// SIMATIC S7-200 SMART project (STEP 7-Micro/WIN SMART), CPU ST40

SYMBOL_TABLE 表格 1
MODBUS_INC       VW100
END_SYMBOL_TABLE

SYMBOL_TABLE 系统符号
Always_On        SM0.0    // 始终接通
END_SYMBOL_TABLE

ORGANIZATION_BLOCK MAIN:OB1
TITLE=程序注释
BEGIN
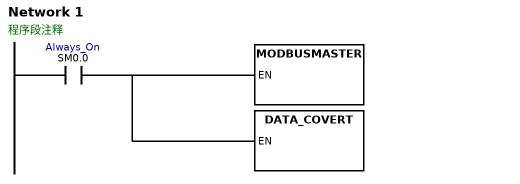
Network 1
// 程序段注释
LD     Always_On:SM0.0
CALL   MODBUSMASTER:SBR41
CALL   DATA_COVERT:SBR4
END_ORGANIZATION_BLOCK

// SBR1: protected block, not included

// SBR2: protected block, not included

// SBR3: protected block, not included

SUBROUTINE_BLOCK DATA_COVERT:SBR4
TITLE=子程序注释
BEGIN
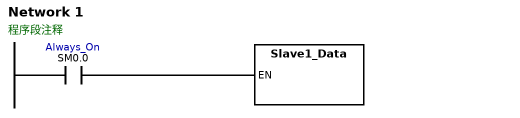
Network 1
// 程序段注释
LD     Always_On:SM0.0
CALL   Slave1_Data:SBR5
END_SUBROUTINE_BLOCK

SUBROUTINE_BLOCK Int_Float:SBR6
TITLE=子程序注释
VAR_INPUT
INPUT:INT;	// LW0 
Coefficient:REAL;	// LD2 
END_VAR
VAR_OUTPUT
OUTPUT:REAL;	// LD6 
END_VAR
VAR
DINT_TEMP:DINT;	// LD10 
REAL_TEMP:REAL;	// LD14 
END_VAR
BEGIN
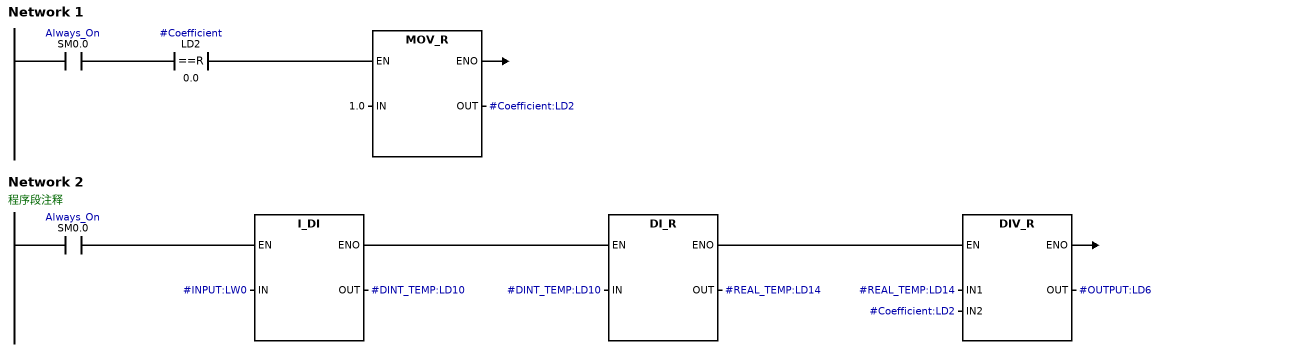
Network 1
LD     Always_On:SM0.0
AR=    #Coefficient:LD2, 0.0
MOVR   1.0, #Coefficient:LD2
Network 2
// 程序段注释
LD     Always_On:SM0.0
ITD    #INPUT:LW0, #DINT_TEMP:LD10
AENO
DTR    #DINT_TEMP:LD10, #REAL_TEMP:LD14
AENO
MOVR   #REAL_TEMP:LD14, #OUTPUT:LD6
/R     #Coefficient:LD2, #OUTPUT:LD6
END_SUBROUTINE_BLOCK

SUBROUTINE_BLOCK Dint_Float:SBR7
TITLE=
VAR_INPUT
INPUT:INT;	// LW0 
Coefficient:REAL;	// LD2 
END_VAR
VAR_OUTPUT
OUT_PUT:REAL;	// LD6 
END_VAR
VAR
DINT_TEMP:DINT;	// LD10 
REAL_TEMP:REAL;	// LD14 
END_VAR
BEGIN
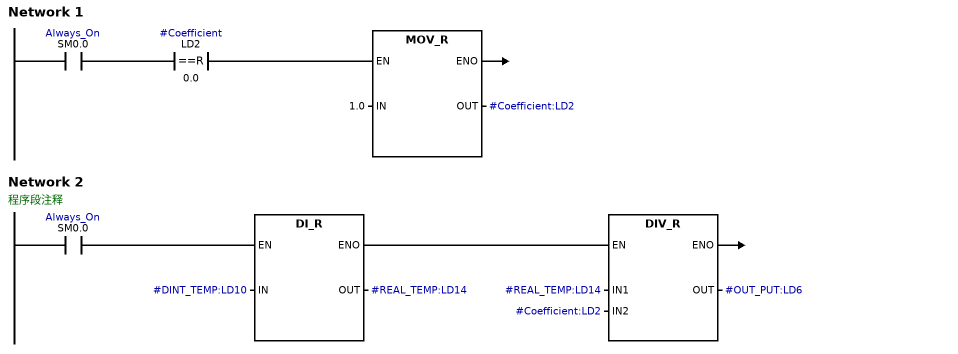
Network 1
LD     Always_On:SM0.0
AR=    #Coefficient:LD2, 0.0
MOVR   1.0, #Coefficient:LD2
Network 2
// 程序段注释
LD     Always_On:SM0.0
DTR    #DINT_TEMP:LD10, #REAL_TEMP:LD14
AENO
MOVR   #REAL_TEMP:LD14, #OUT_PUT:LD6
/R     #Coefficient:LD2, #OUT_PUT:LD6
END_SUBROUTINE_BLOCK

SUBROUTINE_BLOCK MODBUSMASTER:SBR41
TITLE=
VAR
TEMP:BYTE;	// LB0 
TEMP1:BYTE;	// LB1 
TEMP2:BYTE;	// LB2 
TEMP3:BYTE;	// LB3 
TEMP4:BYTE;	// LB4 
TEMP5:BYTE;	// LB5 
TEMP6:BYTE;	// LB6 
TEMPBIT:BOOL;	// L7.0 
TEMPBIT1:BOOL;	// L7.1 
TEMPBIT2:BOOL;	// L7.2 
TEMPBIT3:BOOL;	// L7.3 
TEMPBIT4:BOOL;	// L7.4 
TEMPBIT5:BOOL;	// L7.5 
TEMPBIT6:BOOL;	// L7.6 
END_VAR
BEGIN
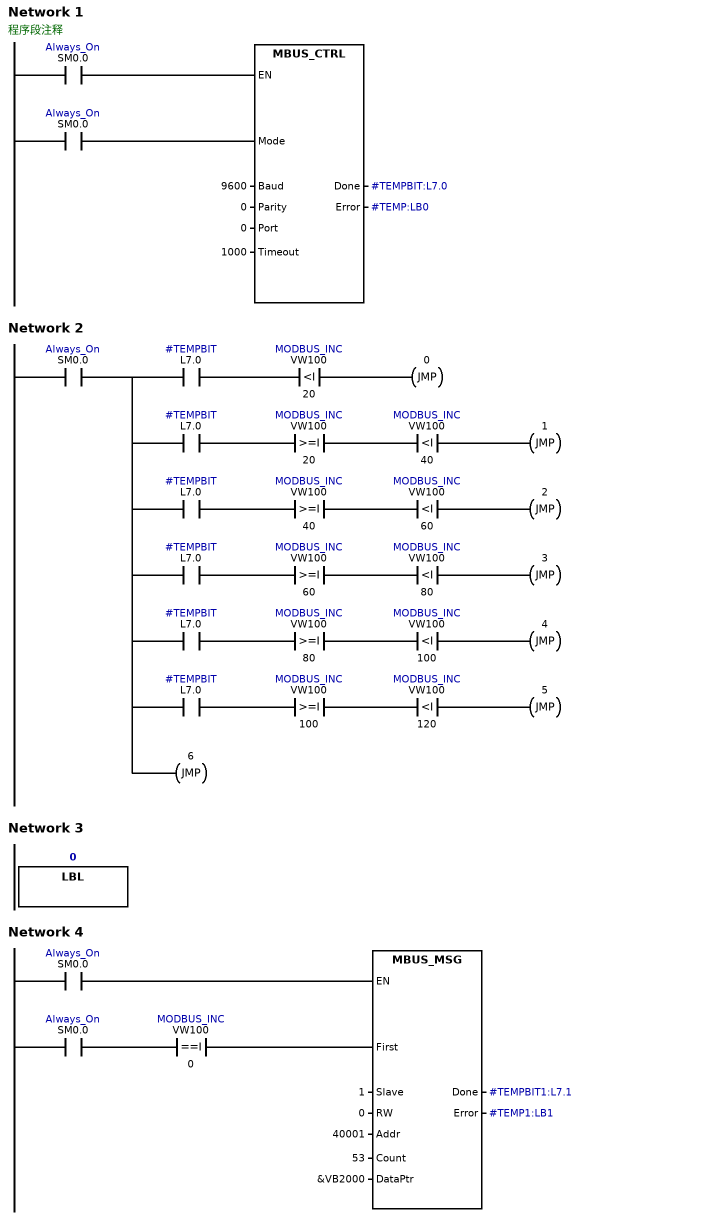
Network 1
// 程序段注释
LD     Always_On:SM0.0
=      L60.0
LD     Always_On:SM0.0
=      L63.7
LD     L60.0
CALL   MBUS_CTRL:SBR1, L63.7, 9600, 0, 0, 1000, #TEMPBIT:L7.0, #TEMP:LB0
Network 2
LD     Always_On:SM0.0
LPS
A      #TEMPBIT:L7.0
AW<    MODBUS_INC:VW100, 20
JMP    0
LRD
A      #TEMPBIT:L7.0
AW>=   MODBUS_INC:VW100, 20
AW<    MODBUS_INC:VW100, 40
JMP    1
LRD
A      #TEMPBIT:L7.0
AW>=   MODBUS_INC:VW100, 40
AW<    MODBUS_INC:VW100, 60
JMP    2
LRD
A      #TEMPBIT:L7.0
AW>=   MODBUS_INC:VW100, 60
AW<    MODBUS_INC:VW100, 80
JMP    3
LRD
A      #TEMPBIT:L7.0
AW>=   MODBUS_INC:VW100, 80
AW<    MODBUS_INC:VW100, 100
JMP    4
LRD
A      #TEMPBIT:L7.0
AW>=   MODBUS_INC:VW100, 100
AW<    MODBUS_INC:VW100, 120
JMP    5
LPP
JMP    6
Network 3
LBL    0
Network 4
LD     Always_On:SM0.0
=      L60.0
LD     Always_On:SM0.0
AW=    MODBUS_INC:VW100, 0
=      L63.7
LD     L60.0
CALL   MBUS_MSG:SBR2, L63.7, 1, 0, 40001, 53, &VB2000, #TEMPBIT1:L7.1, #TEMP1:LB1
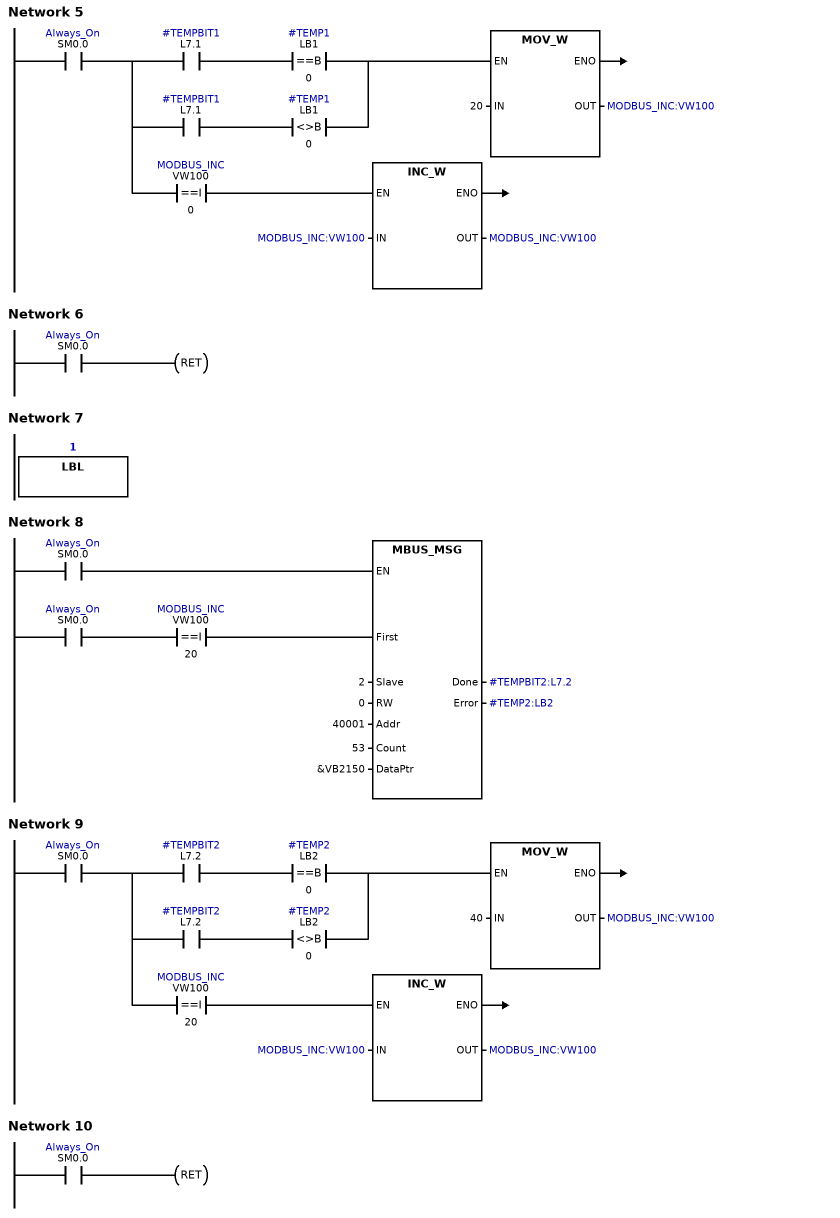
Network 5
LD     Always_On:SM0.0
LPS
LD     #TEMPBIT1:L7.1
AB=    #TEMP1:LB1, 0
LD     #TEMPBIT1:L7.1
AB<>   #TEMP1:LB1, 0
OLD
ALD
MOVW   20, MODBUS_INC:VW100
LPP
AW=    MODBUS_INC:VW100, 0
INCW   MODBUS_INC:VW100
Network 6
LD     Always_On:SM0.0
CRET
Network 7
LBL    1
Network 8
LD     Always_On:SM0.0
=      L60.0
LD     Always_On:SM0.0
AW=    MODBUS_INC:VW100, 20
=      L63.7
LD     L60.0
CALL   MBUS_MSG:SBR2, L63.7, 2, 0, 40001, 53, &VB2150, #TEMPBIT2:L7.2, #TEMP2:LB2
Network 9
LD     Always_On:SM0.0
LPS
LD     #TEMPBIT2:L7.2
AB=    #TEMP2:LB2, 0
LD     #TEMPBIT2:L7.2
AB<>   #TEMP2:LB2, 0
OLD
ALD
MOVW   40, MODBUS_INC:VW100
LPP
AW=    MODBUS_INC:VW100, 20
INCW   MODBUS_INC:VW100
Network 10
LD     Always_On:SM0.0
CRET
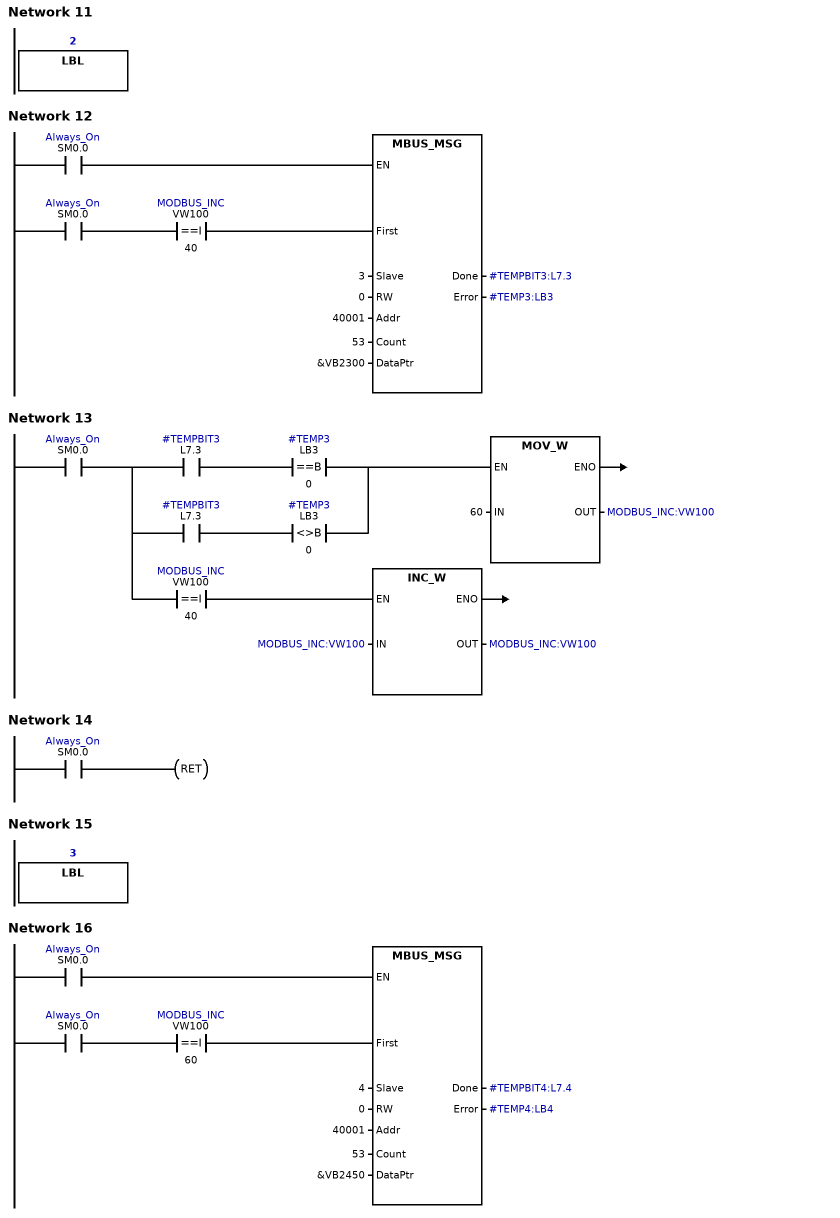
Network 11
LBL    2
Network 12
LD     Always_On:SM0.0
=      L60.0
LD     Always_On:SM0.0
AW=    MODBUS_INC:VW100, 40
=      L63.7
LD     L60.0
CALL   MBUS_MSG:SBR2, L63.7, 3, 0, 40001, 53, &VB2300, #TEMPBIT3:L7.3, #TEMP3:LB3
Network 13
LD     Always_On:SM0.0
LPS
LD     #TEMPBIT3:L7.3
AB=    #TEMP3:LB3, 0
LD     #TEMPBIT3:L7.3
AB<>   #TEMP3:LB3, 0
OLD
ALD
MOVW   60, MODBUS_INC:VW100
LPP
AW=    MODBUS_INC:VW100, 40
INCW   MODBUS_INC:VW100
Network 14
LD     Always_On:SM0.0
CRET
Network 15
LBL    3
Network 16
LD     Always_On:SM0.0
=      L60.0
LD     Always_On:SM0.0
AW=    MODBUS_INC:VW100, 60
=      L63.7
LD     L60.0
CALL   MBUS_MSG:SBR2, L63.7, 4, 0, 40001, 53, &VB2450, #TEMPBIT4:L7.4, #TEMP4:LB4
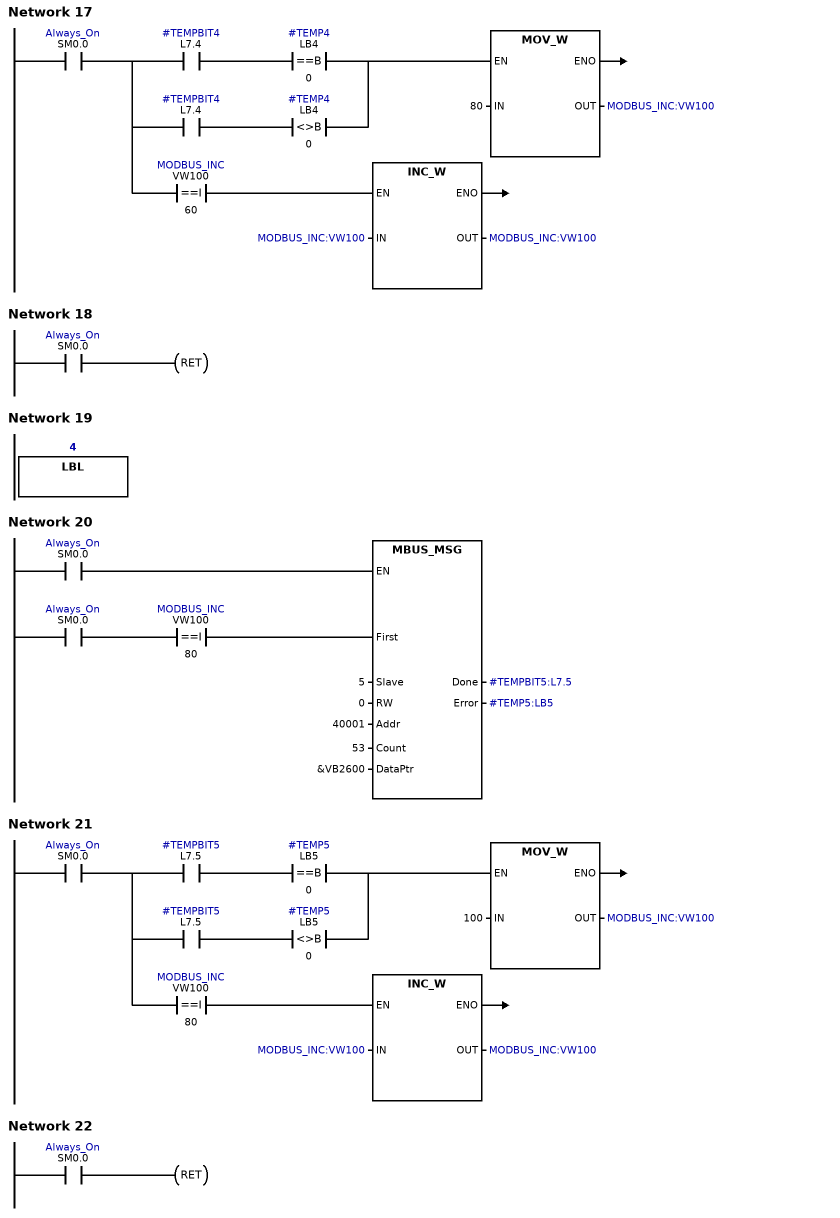
Network 17
LD     Always_On:SM0.0
LPS
LD     #TEMPBIT4:L7.4
AB=    #TEMP4:LB4, 0
LD     #TEMPBIT4:L7.4
AB<>   #TEMP4:LB4, 0
OLD
ALD
MOVW   80, MODBUS_INC:VW100
LPP
AW=    MODBUS_INC:VW100, 60
INCW   MODBUS_INC:VW100
Network 18
LD     Always_On:SM0.0
CRET
Network 19
LBL    4
Network 20
LD     Always_On:SM0.0
=      L60.0
LD     Always_On:SM0.0
AW=    MODBUS_INC:VW100, 80
=      L63.7
LD     L60.0
CALL   MBUS_MSG:SBR2, L63.7, 5, 0, 40001, 53, &VB2600, #TEMPBIT5:L7.5, #TEMP5:LB5
Network 21
LD     Always_On:SM0.0
LPS
LD     #TEMPBIT5:L7.5
AB=    #TEMP5:LB5, 0
LD     #TEMPBIT5:L7.5
AB<>   #TEMP5:LB5, 0
OLD
ALD
MOVW   100, MODBUS_INC:VW100
LPP
AW=    MODBUS_INC:VW100, 80
INCW   MODBUS_INC:VW100
Network 22
LD     Always_On:SM0.0
CRET
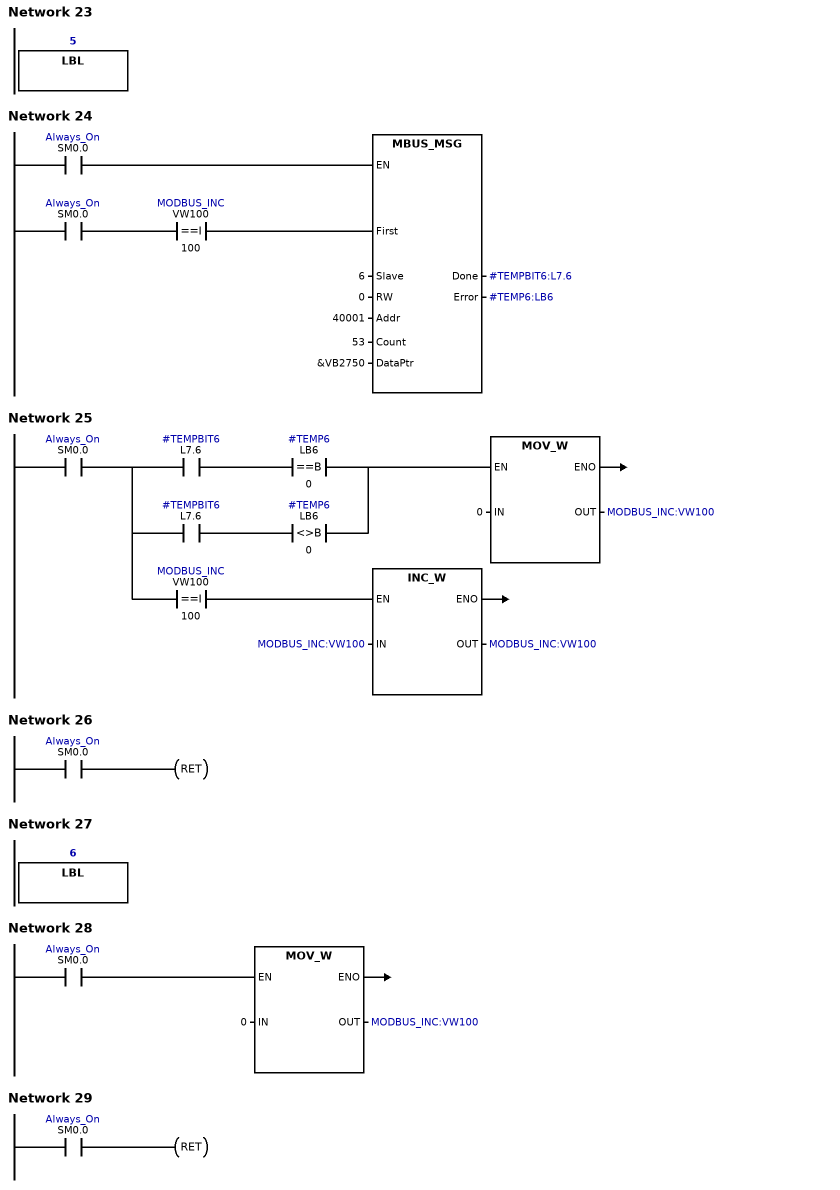
Network 23
LBL    5
Network 24
LD     Always_On:SM0.0
=      L60.0
LD     Always_On:SM0.0
AW=    MODBUS_INC:VW100, 100
=      L63.7
LD     L60.0
CALL   MBUS_MSG:SBR2, L63.7, 6, 0, 40001, 53, &VB2750, #TEMPBIT6:L7.6, #TEMP6:LB6
Network 25
LD     Always_On:SM0.0
LPS
LD     #TEMPBIT6:L7.6
AB=    #TEMP6:LB6, 0
LD     #TEMPBIT6:L7.6
AB<>   #TEMP6:LB6, 0
OLD
ALD
MOVW   0, MODBUS_INC:VW100
LPP
AW=    MODBUS_INC:VW100, 100
INCW   MODBUS_INC:VW100
Network 26
LD     Always_On:SM0.0
CRET
Network 27
LBL    6
Network 28
LD     Always_On:SM0.0
MOVW   0, MODBUS_INC:VW100
Network 29
LD     Always_On:SM0.0
CRET
END_SUBROUTINE_BLOCK
